(* CODESYS project SortingByWeight.project

Project tree, tasks and I/O mapping:
  Device : CODESYS Control Win V3, 3S - Smart Software Solutions GmbH, order no. 305021, version 3.5.7.20
    application Application
      libraries: Standard, * (System)
      task MainTask (cyclic, interval t#20ms, priority 1) calls Main
      program Main [ST]: Station_Call, Outputs_Management, Stop_Management
      global variables GVL_Sensors_And_Actuators
      Symbols
      data type Enum_Motor_Status
      Stations/
        program Entry_Station [ST]
        program Right_Exit_Station [ST]
        program Left_Exit_Station [ST]
        program Front_Exit_Station [ST]
        program Weighing_Station [ST]
        program Load_Scale_Station [ST]
      global variables Var_System
*)

// Device/Application/Enum_Motor_Status
{attribute 'strict'}
TYPE Enum_Motor_Status :
(
	Stopped :=	0,
	Star :=	1,
	Delta := 2,
	Failure	:=	3
);
END_TYPE

// Device/Application/GVL_Sensors_And_Actuators
VAR_GLOBAL
	
	// Digital Inputs
	Auto				:BOOL; // Auto mode switch = 0
	Manual				:BOOL; // Manual mode switch "NC" = 1
	Reset				:BOOL; // reset button
	Start				:BOOL; // start button
	Stop				:BOOL; // stop button "NC" = 1
	Emergency_Stop		:BOOL; // emergency stop "NC" = 1
	Factory_Reset		:BOOL; // Bit to reset factory scene
	Factory_Run			:BOOL; // bit to start factory scene
	At_Scale_Entry		:BOOL; // at scale entry sensor "NC" = 1
	At_Scale			:BOOL; // at scale sensor "NC" = 1
	At_Scale_Exit		:BOOL; // at scale exit sensor 
	At_Left_Entry		:BOOL; // at left entry sensor 
	At_Forward_Entry	:BOOL; // at forward entry sensor
	At_Right_Entry		:BOOL; // at right entry sensor
	At_Exit_Left		:BOOL; // at exit left sensor "NC" = 1
	At_Exit_Front		:BOOL; // at exit front sensor "NC" = 1
	At_Exit_Right		:BOOL; // at exit right sensor "NC" = 1

	
	
	// Analog Inputs
	Weight				:REAL; // weighing sensor
	Left_Count			:INT;  // counter sensor for boxes sent to left 
	Right_Count			:INT;  // counter sensor for boxes sent to right 
	Front_Count			:INT;  // counter sensor for boxes sent to front 
	
	
	// Digital Outputs
	Entry_Convey		:BOOL; // entry conveyor motor
	Front_Convey		:BOOL; // front conveyor motor
	Right_Convey		:BOOL; // right conveyor motor
	Left_Convey			:BOOL; // left conveyor motor
	Load_Scale_Convey	:BOOL; // product on scale actuator
	Send_Left			:BOOL; // box selector send to left
	Send_Right			:BOOL; // box selector send to right
	Send_Front			:BOOL; // box selector send to front
	System_Active_Led	:BOOL;
	System_Stopped_Led	:BOOL;
	

END_VAR

// Device/Application/Var_System
VAR_GLOBAL
	// Inputs
	System_Active		:BOOL;
	Soft_Stop_Active	:BOOL;
	
	// Counter Var
	Right_Counter		:INT :=0;
	Left_Counter 		:INT :=0;
	Front_Counter		:INT :=0;
	
	// Timers
	Scale_Timer			:TON;
	Load_Timer			:TON;				
	
	// Timer Var
	Weighin_Time		:TIME := T#1S;	
	Time_Weighing		:TIME; 				
	Load_Time			:TIME := T#2.5S;	
	Time_Weighing_Elap	:TIME;
	Time_Scale_Elap		:TIME;
	
	// OutPut memories
	M_Entry_Convey		:BOOL;
	M_Front_Convey		:BOOL;
	M_Right_Convey		:BOOL;
	M_Left_Convey		:BOOL;
	M_Load_Convey		:BOOL;
	M_Box_To_Left		:BOOL;
	M_Box_To_Right		:BOOL;
	M_Box_To_Front		:BOOL;
	
END_VAR

// Device/Application/Main
PROGRAM Main
VAR
	Ons_Start_Entry					:R_TRIG;
END_VAR

(*
* File: Main Program
* Author: Jaime Calvente Mieres
* Date: 12-08-2022
* Description: Main program to manage the Stations,
* outputs and Start/Stop management. 
*)

(*
 * Systeme will be active if Start button is pressed 
 * and Stop and Emergency stop aren't "NC". 
 * When the system is active this program will call the actions
 * to execute the logic programmed in them. 
*)

// One shot Start
Ons_Start_Entry(CLK:= Start);

// Action calls
Station_Call();
Outputs_Management();
Stop_Management();

// System bit activation
IF Ons_Start_Entry.Q AND Stop AND Emergency_Stop THEN
	System_Active := TRUE;
	Soft_Stop_Active := FALSE;
END_IF

ACTION Station_Call:
(*
* File: Station Call
* Author: Jaime Calvente Mieres
* Date: 12-08-2022
* Description: Action to Call the different stations of the plant. 
*)


(* Station calls to make the program modular,
eac station will be call one after the other. *)
Entry_Station();
Load_Scale_Station();
Weighing_Station();
Right_Exit_Station();
Left_Exit_Station();
Front_Exit_Station();
END_ACTION

ACTION Outputs_Management:
(*
* File: Station Call
* Author: Jaime Calvente Mieres
* Date: 12-08-2022
* Description: Action to map the outputs with the programm variables. 
*)

(*
 * Mapping of the system outputs to system var
 * to make the implementation clearer and more efficient
 *)

// Entry conveyor coil activation
Entry_Convey := M_Entry_Convey;

// Load Scale conveyor coil activation
Load_Scale_Convey := M_Load_Convey;
 
// Send Box to Front box selector
Send_Front := M_Box_To_Front OR 
				M_Box_To_Left OR 
				M_Box_To_Right;
				
// Front conveyor coil activation
Front_Convey := M_Front_Convey;				
				
// Send Box to Left box selector				
Send_Left := M_Box_To_Left;

// Left conveyor coil activation
Left_Convey := M_Left_Convey;

// Send Box to Right box selector
Send_Right := M_Box_To_Right;

// Right conveyor coil activation
Right_Convey :=  M_Right_Convey;


// System Leds activation
System_Active_Led := System_Active;
System_Stopped_Led := Soft_Stop_Active OR NOT Emergency_Stop;
END_ACTION

ACTION Stop_Management:
(*
* File: Stop Management
* Author: Jaime Calvente Mieres
* Date: 14-08-2022
* Description: Action to Manage the Emergency Stop and Soft Stopt management. 
*)

// If Emergency Stop is pressed Reset the system
IF NOT Emergency_Stop THEN
	
	System_Active 		:= FALSE;
	Entry_Convey 		:= FALSE;
	Load_Scale_Convey 	:= FALSE;
	Left_Convey 		:= FALSE;
	Right_Convey 		:= FALSE;
	Front_Convey 		:= FALSE;
	M_Box_To_Front 		:= FALSE;
	M_Box_To_Left 		:= FALSE;
	M_Box_To_Right 		:= FALSE;
	M_Right_Convey 		:= FALSE;
	M_Entry_Convey 		:= FALSE;
	M_Load_Convey 		:= FALSE;
	Load_Timer.IN 		:= FALSE;
	Scale_Timer.IN 		:= FALSE;
	M_Front_Convey 		:= FALSE;
	M_Left_Convey 		:= FALSE;
	// Counters Reset
	Right_Counter 		:= 0;
	Right_Count			:= 0;
	Left_Counter 		:= 0;
	Left_Count			:= 0;
	Front_Counter 		:= 0;
	Front_Count			:= 0;
	
END_IF


// If Stop button Reset System and Activate Soft_Stop bit
IF NOT Stop THEN
	Soft_Stop_Active := TRUE;
	System_Active := FALSE;
END_IF
END_ACTION

END_PROGRAM

// Device/Application/Stations/Entry_Station
PROGRAM Entry_Station
VAR
	Ons1_Box_Leaving_Scale		:F_TRIG;
	Ons2_Box_Stopped_At_Scales	:F_TRIG;
END_VAR

(*
* File: Entry Conveyor
* Author: Jaime Calvente Mieres
* Date: 12-08-2022
* Description: Program to control the box entry conveyor belt. 
*)

(* Conditions to activate the Entry conveyor *)
IF System_Active THEN
	
	// One shot calls
	Ons1_Box_Leaving_Scale(CLK := At_Scale);
	
	(* Entry conveyor activation if the system is Activated *)
	// If not box at scale sensor or Scale sensor 
	IF (NOT At_Scale AND NOT At_Scale_Entry) OR
		(Ons2_Box_Stopped_At_Scales.Q AND At_Scale_Entry) OR
		Ons1_Box_Leaving_Scale.Q THEN
		M_Entry_Convey := TRUE ;	
	END_IF
	
	(*If scale sensor and One shot of At Scale entry
	 sensor Stop Entry conveyor*)
	IF At_Scale THEN
		M_Entry_Convey := FALSE;
	END_IF
	
END_IF


(* Conditions to Re-Start the program after
 a soft stop *)
Ons2_Box_Stopped_At_Scales(CLK := Soft_Stop_Active);
IF Soft_Stop_Active AND M_Entry_Convey AND (At_Scale OR At_Scale_Entry) THEN
	M_Entry_Convey := FALSE;
END_IF

END_PROGRAM

// Device/Application/Stations/Load_Scale_Station
PROGRAM Load_Scale_Station
VAR
	Ons3_At_Scale			:R_TRIG;
	Ons4_Timer_Out			:R_TRIG;
	Ons5_Box_At_Entry		:R_TRIG;
END_VAR

(*
* File: Load Scale Station
* Author: Jaime Calvente Mieres
* Date: 13-08-2022
* Description: Program to control the box loading into the Scale. 
*)


(*
 * If system is active allow to load boxes into the scale
 * and set the timer to allow weighing time. 
 *)
IF System_Active THEN
	// One shot declarations
	Ons3_At_Scale(CLK := At_Scale);
	Ons4_Timer_Out(CLK := Load_Timer.Q);
	Ons5_Box_At_Entry(CLK := At_Scale_Entry);
	
	// Timer instantiation
	Load_Timer(IN := (At_Scale AND NOT Soft_Stop_Active) , PT := Load_Time, ET => Time_Weighing_Elap);
	
	(* Load conveyor activation when not box at scale AND 
	at scale entry OR timer output is active *)
	IF (Ons5_Box_At_Entry.Q AND NOT At_Scale) OR Ons4_Timer_Out.Q THEN
		M_Load_Convey := TRUE;
	END_IF
	
	// If box at Scale sensor deactivate conveyor and SET timer
	IF Ons3_At_Scale.Q OR Soft_Stop_Active AND (M_Load_Convey AND At_Scale) THEN
		M_Load_Convey := FALSE;
	END_IF
	
END_IF

(* Conditions to Re-Start the program after
 a soft stop *)
IF Soft_Stop_Active AND M_Load_Convey AND At_Scale THEN
	M_Load_Convey := FALSE;
END_IF

END_PROGRAM

// Device/Application/Stations/Weighing_Station
PROGRAM Weighing_Station
VAR
	Ons6_Front_Entry			:F_TRIG;
	Ons7_Left_Entry				:F_TRIG;
	Ons8_Right_Entry			:F_TRIG;
END_VAR

(*
* File: Weighing Station
* Author: Jaime Calvente Mieres
* Date: 14-08-2022
* Description: Program to control the weight management process of boxes
* and paht selection depending on size. 
*)


(*
 * If system active and there is a box at scale sensor then start weighing 
 * the boxes and set a weighin time. When the time has passed, the output of
 * the timer will free up the path selection to exit the boxes. 
 *)
IF System_Active THEN
	// One shot instances
	Ons6_Front_Entry(CLK := At_Forward_Entry);
	Ons7_Left_Entry(CLK := At_Left_Entry);
	Ons8_Right_Entry(CLK:= At_Right_Entry);
	
	// Timer instantiation
	Scale_Timer(IN := (At_Scale AND NOT Soft_Stop_Active), PT :=  Weighin_Time, ET => Time_Scale_Elap);
	
	(* Box Path selection by weight when timer out is "On" *)
	IF Scale_Timer.Q THEN
		// Large box size to Front
		IF (Weight >= 5.0) AND NOT (M_Box_To_Right OR M_Box_To_Left)  THEN
			M_Box_To_Front := TRUE;
		// Medium size box to Right
		ELSIF (Weight >= 3.5 AND Weight < 5.0) AND NOT (M_Box_To_Front OR M_Box_To_Left) THEN
			M_Box_To_Right := TRUE;
		// Small size box to Left	
		ELSIF (Weight >= 1.5 AND Weight < 3.5) AND NOT (M_Box_To_Front OR M_Box_To_Right) THEN
			M_Box_To_Left := TRUE;	
		END_IF
	END_IF

	(* Box Path selector Deactivations *)
	// Front path reset
	IF Ons6_Front_Entry.Q THEN
		M_Box_To_Front := FALSE;
	END_IF
	// Letf path reset
	IF Ons7_Left_Entry.Q THEN
		M_Box_To_Left := FALSE;	
	END_IF
	// Right path reset
	IF Ons8_Right_Entry.Q THEN
		M_Box_To_Right := FALSE;
	END_IF
		
(* If not system active due to an emergency stop
 or a soft stop, deactivate the box selector and 
 reset the timer. *)	
ELSE
	Scale_Timer.IN := FALSE;
	M_Box_To_Front := FALSE;
	M_Box_To_Left := FALSE;	
	M_Box_To_Right := FALSE;
END_IF

END_PROGRAM

// Device/Application/Stations/Right_Exit_Station
PROGRAM Right_Exit_Station
VAR
	Box_At_Right_Convey				:BOOL;
	Ons13_Right_Entry				:R_TRIG;
	Ons14_Exit_Right				:R_TRIG;
	Ons15_Re_Energize				:F_TRIG;
	Ons16_Counter					:R_TRIG;
END_VAR

(*
* File: Right Exit Conveyor
* Author: Jaime Calvente Mieres
* Date: 13-08-2022
* Description: Program to control the right exit path of the boxes. 
*)


(* 
 * If the systme is active and sensor at left entry
 * fires up, activate the conveyor and count one box.
 * If the Exit sensor Negative edge detects a box,
 * decrease the counter by one and check if conveyor
 * needs to be stopped or not. 
 *)
IF System_Active THEN
	
	// One shot call
	Ons13_Right_Entry(CLK:= At_Right_Entry);
	Ons14_Exit_Right(CLK := At_Exit_Right);
	Ons16_Counter(CLK := At_Right_Entry);
	
	// Convey Activation conditions
	IF Ons15_Re_Energize.Q AND ( Right_Counter <> 0 OR At_Right_Entry) OR Ons13_Right_Entry.Q  THEN
		M_Right_Convey := TRUE;
	END_IF

	// Set box at scale and increment counter
	IF Ons16_Counter.Q THEN
		//Box_At_Right_Convey := TRUE;
		Right_Count := Right_Count +1;
		Right_Counter := Right_Counter +1;
	END_IF
	
	// Counter decrement and Box at convey deactivation
	IF Ons14_Exit_Right.Q THEN
		//Box_At_Right_Convey := FALSE;
		// Check the counter to decrease it
		IF Right_Counter <> 0 THEN
			Right_Counter := Right_Counter - 1;
		// Check the counter to deactivate the Convey
		ELSIF Right_Counter = 0 THEN
			M_Right_Convey := FALSE;	
		END_IF
	END_IF	
	
END_IF


(* Conditions to Re-Start the program after
 a soft stop *)
Ons15_Re_Energize(CLK := Soft_Stop_Active);
IF Soft_Stop_Active THEN
	M_Right_Convey := FALSE;
END_IF

END_PROGRAM

// Device/Application/Stations/Left_Exit_Station
PROGRAM Left_Exit_Station
VAR
	Box_At_Left_Convey							:BOOL;
	Ons9_Left_Entry								:R_TRIG;
	Ons10_Exit_Left								:R_TRIG;
	Ons11_Re_Energize							:F_TRIG;
	Ons12_Box_counter							:R_TRIG;
END_VAR

(*
* File: Left Exit Conveyor
* Author: Jaime Calvente Mieres
* Date: 13-08-2022
* Description: Program to control the left exit path of the boxes.
*)


(* 
 * If the systme is active and sensor at left entry
 * fires up, activate the conveyor and count one box.
 * If the Exit sensor Negative edge detects a box,
 * decrease the counter by one and check if conveyor
 * needs to be stopped or not. 
 *)
IF System_Active THEN
	// One shots
	Ons9_Left_Entry(CLK:= At_Left_Entry);
	Ons10_Exit_Left(CLK := At_Exit_Left);
	Ons12_Box_counter(CLK := At_Left_Entry);
	
	// Convey Activation conditions
	IF Ons11_Re_Energize.Q AND (Left_Counter <> 0 OR At_Left_Entry) OR Ons9_Left_Entry.Q THEN
		M_Left_Convey := TRUE;
	END_IF
	
	// Set box at convy and increment counter
	IF Ons12_Box_counter.Q THEN
		//Box_At_Left_Convey := TRUE;
		Left_Counter := Left_Counter + 1;
		Left_Count := Left_Count + 1;
	END_IF

	// Counter decrement and Box at convey deactivation
	IF Ons10_Exit_Left.Q THEN
		//Box_At_Left_Convey := FALSE;
		// Check the counter to decrease the counter
		IF Left_Counter <> 0 THEN
			Left_Counter := Left_Counter - 1;
		// Check the counter to deactivate the Convey
		ELSIF Left_Counter = 0 THEN
			M_Left_Convey := FALSE;
		END_IF	
	END_IF
	
END_IF

(* Conditions to Re-Start the program after
 a soft stop *)
Ons11_Re_Energize(CLK := Soft_Stop_Active);
IF Soft_Stop_Active THEN
	M_Left_Convey := FALSE;
END_IF

END_PROGRAM

// Device/Application/Stations/Front_Exit_Station
PROGRAM Front_Exit_Station
VAR
	Box_At_Front_Convey						:BOOL;
	Ons17_Forward_Entry						:R_TRIG;
	Ons18_Exit_Front						:R_TRIG;
	Ons19_Re_Energize						:F_TRIG;
	Ons20_Counter							:R_TRIG;
END_VAR

(*
* File: Front Exit Conveyor
* Author: Jaime Calvente Mieres
* Date: 13-08-2022
* Description: Program to control the front exit path of the boxes.
*)


(* 
 * If the systme is active and sensor at left entry
 * fires up, activate the conveyor and count one box.
 * If the Exit sensor Negative edge detects a box,
 * decrease the counter by one and check if conveyor
 * needs to be stopped or not. 
 *)
IF System_Active THEN
	// One shots
	Ons17_Forward_Entry(CLK:= At_Forward_Entry);
	Ons18_Exit_Front(CLK := At_Exit_Front);
	Ons20_Counter(CLK := At_Forward_Entry);
	
	// Convey Activation conditions
	IF Ons19_Re_Energize.Q AND (Front_Counter <> 0 OR At_Forward_Entry) OR Ons17_Forward_Entry.Q THEN
		// Activate conveyor,
		M_Front_Convey := TRUE;
	END_IF
	
	// Set box at convey and increment counter
	IF Ons20_Counter.Q THEN
		//Box_At_Front_Convey := TRUE; 
		Front_Counter := Front_Counter + 1;
		Front_Count := Front_Count + 1;
	END_IF
	
	// Counter decrement and Box at convey deactivation
	IF Ons18_Exit_Front.Q THEN
		//Box_At_Front_Convey := FALSE; 
		// Check the counter to decrease the counter
		IF Front_Counter <> 0 THEN
			Front_Counter := Front_Counter - 1;
		// Check the counter to deactivate the Convey
		ELSIF Front_Counter = 0 THEN
			M_Front_Convey := FALSE;		
		END_IF
	END_IF
	
END_IF

(* Conditions to Re-Start the program after
 a soft stop *)
Ons19_Re_Energize(CLK := Soft_Stop_Active);
IF Soft_Stop_Active THEN
	M_Front_Convey := FALSE;
END_IF

END_PROGRAM
